INTERFACE I_State

METHOD PUBLIC Handle : BOOL
END_METHOD

END_INTERFACE

(* stored: Version 1.1.0.1, ProductVersion 3.1.4024.3
   Itf I_State: Id {8e73192b-d2e1-43c8-ad43-720eb715c850}
   Method Handle: Id {d70289f2-db71-41b6-941b-611f697e3b7b} *)
